      "DEV_Spk-000CDL:Cryo-PT-91_iDB" (EPICSToPLCLength:=15,
      EPICSToPLCDataBlockOffset:=572,
      PLCToEPICSLength:=25,
      PLCToEPICSDataBlockOffset:=1327);

        //********************************************
        // Device name: Spk-000CDL:Cryo-PT-92
        // Device type: ICS_PT_mbar
        //********************************************

      "DEV_Spk-000CDL:Cryo-PT-92_iDB" (EPICSToPLCLength:=15,
      EPICSToPLCDataBlockOffset:=587,
      PLCToEPICSLength:=25,
      PLCToEPICSDataBlockOffset:=1352);

        //********************************************
        // Device name: Spk-000CDL:Cryo-PT-93
        // Device type: ICS_PT_mbar
        //********************************************

      "DEV_Spk-000CDL:Cryo-PT-93_iDB" (EPICSToPLCLength:=15,
      EPICSToPLCDataBlockOffset:=602,
      PLCToEPICSLength:=25,
      PLCToEPICSDataBlockOffset:=1377);

        //********************************************
        // Device name: Spk-000CDL:Cryo-PT-94
        // Device type: ICS_PT_mbar
        //********************************************

      "DEV_Spk-000CDL:Cryo-PT-94_iDB" (EPICSToPLCLength:=15,
      EPICSToPLCDataBlockOffset:=617,
      PLCToEPICSLength:=25,
      PLCToEPICSDataBlockOffset:=1402);

        //********************************************
        // Device name: Spk-000CDL:Cryo-PT-95
        // Device type: ICS_PT_mbar
        //********************************************

      "DEV_Spk-000CDL:Cryo-PT-95_iDB" (EPICSToPLCLength:=15,
      EPICSToPLCDataBlockOffset:=632,
      PLCToEPICSLength:=25,
      PLCToEPICSDataBlockOffset:=1427);

        //********************************************
        // Device name: Spk-000CDL:Vac-VGC-071
        // Device type: ICS_PT_mbar
        //********************************************

      "DEV_Spk-000CDL:Vac-VGC-071_iDB" (EPICSToPLCLength:=15,
      EPICSToPLCDataBlockOffset:=647,
      PLCToEPICSLength:=25,
      PLCToEPICSDataBlockOffset:=1452);

        //********************************************
        // Device name: Spk-000CDL:Vac-VGP-070
        // Device type: ICS_PT_mbar
        //********************************************

      "DEV_Spk-000CDL:Vac-VGP-070_iDB" (EPICSToPLCLength:=15,
      EPICSToPLCDataBlockOffset:=662,
      PLCToEPICSLength:=25,
      PLCToEPICSDataBlockOffset:=1477);
END_FUNCTION
DATA_BLOCK "EPICS_DebuggerResult"
{ S7_Optimized_Access := 'TRUE' }
VERSION : 0.1
NON_RETAIN
   VAR
      EPICS_Debugger_UtilitiesCall : String;   // PLCFactory Utilities call status
      EPICS_Debugger_DeviceCalls : String;   // PLCFactory DeviceCalls status
      EPICS_Debugger_IOCHash : String;   // EPICS IOC Hash vs. PLCFactory Hash
      EPICS_Debugger_ModBusHeartBeat : String;   // EPICS IOC Modbus (IOC->PLC) communication status
      EPICS_Debugger_S7Connection : String;   // EPICS IOC S7 TCP (PLC->IOC) communication status
      EPICS_Debugger_EPICS_GeneralState : String;   // Main status of the EPICS IOC communication
      EPICS_S7Port : Int;   // Actual TCP port that has been opened by the PLC
      EPICS_ModbusPort : Int;   // Actual ModBusTCP port that has been opened by the PLC
      EPICS_PLC_EthernetInterface : UInt;   // The currently used HW Identifer of the Ethernet Port on the PLC dedicated to EPICS
      EPICS_PayloadSize_InBytes : UInt;   // The currently configured payload size in bytes
      EPICS_PLC_Hash : DInt;   // The PLC Hash
      EPICS_PLCFactory_Version : String;   // The PLCFactory version that was used to generate the PLC code
      EPICS_CommunicationOK : Bool;   // Overall EPICS communication is OK
   END_VAR

BEGIN

END_DATA_BLOCK
FUNCTION_BLOCK "EPICS_DebuggerFB"
{ S7_Optimized_Access := 'TRUE' }
VERSION : 0.1
   VAR
      CheckUtilitiesTON {OriginalPartName := 'IEC_TIMER'; LibVersion := '1.0'; ExternalAccessible := 'False'; ExternalVisible := 'False'; ExternalWritable := 'False'} : TON_TIME;
      UtilSquareErrorTON { ExternalAccessible := 'False'; ExternalVisible := 'False'; ExternalWritable := 'False'} : Bool;
      CheckUtilitiesTON2 {OriginalPartName := 'IEC_TIMER'; LibVersion := '1.0'; ExternalAccessible := 'False'; ExternalVisible := 'False'; ExternalWritable := 'False'} : TON_TIME;
      UtilSquareErrorTON2 { ExternalAccessible := 'False'; ExternalVisible := 'False'; ExternalWritable := 'False'} : Bool;
      ModBus_TON {OriginalPartName := 'IEC_TIMER'; LibVersion := '1.0'; ExternalAccessible := 'False'; ExternalVisible := 'False'; ExternalWritable := 'False'} : TON_TIME;
      ModBus_wordsave { ExternalAccessible := 'False'; ExternalVisible := 'False'; ExternalWritable := 'False'} : Word;
   END_VAR
   VAR DB_SPECIFIC
      Helper_String { ExternalAccessible := 'False'; ExternalVisible := 'False'; ExternalWritable := 'False'} : String;
      Helper_String_Array { ExternalAccessible := 'False'; ExternalVisible := 'False'; ExternalWritable := 'False'} AT Helper_String : Struct
         String_Maximal { ExternalAccessible := 'False'; ExternalVisible := 'False'; ExternalWritable := 'False'} : Byte;
         String_Actual { ExternalAccessible := 'False'; ExternalVisible := 'False'; ExternalWritable := 'False'} : Byte;
         StringValueArray { ExternalAccessible := 'False'; ExternalVisible := 'False'; ExternalWritable := 'False'} : Array[0..15] of Byte;
      END_STRUCT;
   END_VAR
   VAR
      S7ConnTON {OriginalPartName := 'IEC_TIMER'; LibVersion := '1.0'; ExternalAccessible := 'False'; ExternalVisible := 'False'; ExternalWritable := 'False'} : TON_TIME;
   END_VAR

   VAR_TEMP
      AllOK { ExternalAccessible := 'False'; ExternalVisible := 'False'; ExternalWritable := 'False'} : Bool;
      i : Int;
      ModBusOK : Bool;
      S7OK : Bool;
   END_VAR


BEGIN
	//Author: Miklos Boros (miklos.boros@esss.se), Copyrigth 2017-2020 by European Spallation Source, Lund
	//This block was generated by PLCFactory
	//Description: This FB checks the EPICS configuration and outputs the result into EPICS_DebuggerResult.

	//DO NOT Modify this block!!!

	//AllOK will be evaluated in this code and passed to the EPICS_CommunicationOK signal that can be used by the PLC logic
	#AllOK := TRUE;

	#CheckUtilitiesTON(IN:="Utilities".Square_100ms,
	                   PT:=T#200ms,
	                   Q=>#UtilSquareErrorTON);

	#CheckUtilitiesTON2(IN := NOT "Utilities".Square_100ms,
	                   PT := T#200ms,
	                   Q => #UtilSquareErrorTON2);


	#ModBus_TON(IN := #ModBus_wordsave = "EPICSToPLC"."Word"[2],
	            PT := T#5s);


     "EPICS_DebuggerResult".#EPICS_PayloadSize_InBytes := 3004;
     "EPICS_DebuggerResult".#EPICS_PLC_Hash := 457744924;
     "EPICS_DebuggerResult".#EPICS_PLCFactory_Version := 'fb3b582a9a66e37ff877560bc4f23ab7654f4230';

	IF ("Utilities".AlwaysOn = FALSE) THEN
	    "EPICS_DebuggerResult".#EPICS_Debugger_UtilitiesCall := 'ERROR: FunctionBlock: "_UilitiesFB" is called with a wrong InstanceDB. Call it with the existing iDB named: "Utilities" AND check if the System Memory bits and the System Clock byte is enabled!';
         #AllOK := FALSE;
	ELSE
	    IF (#UtilSquareErrorTON OR #UtilSquareErrorTON2) THEN
	        "EPICS_DebuggerResult".#EPICS_Debugger_UtilitiesCall := 'ERROR: FunctionBlock: "_UilitiesFB" is called with a wrong InstanceDB. Call it with the existing iDB named: "Utilities" AND check if the System Memory bits and the System Clock byte is enabled!';
             #AllOK := FALSE;
	    ELSE
	        "EPICS_DebuggerResult".#EPICS_Debugger_UtilitiesCall := 'OK: EPICS Utilities works as expected.';

	    END_IF;
	END_IF;

	IF ("Utilities".EPICS_Device_calls_precessed) THEN
	    "EPICS_DebuggerResult".#EPICS_Debugger_DeviceCalls := 'OK: "EPICS_device_calls" is called as expected.';
	ELSE
	    "EPICS_DebuggerResult".#EPICS_Debugger_DeviceCalls := 'ERROR: "EPICS_device_calls" is not called in OB1!';
         #AllOK := FALSE;
	END_IF;

	IF (("EPICSToPLC"."Word"[0] = "PLCToEPICS"."Word"[0]) AND ("EPICSToPLC"."Word"[1] = "PLCToEPICS"."Word"[1])) THEN
	    "EPICS_DebuggerResult".#EPICS_Debugger_IOCHash := 'OK: IOC and PLC hash are equal.';
	ELSE
	    "EPICS_DebuggerResult".#EPICS_Debugger_IOCHash := 'ERROR: IOC and PLC hash are NOT equal!';
         #AllOK := FALSE;
	END_IF;

	IF (#ModBus_TON.Q) THEN
	    "EPICS_DebuggerResult".#EPICS_Debugger_ModBusHeartBeat := 'ERROR: The IOC is not sending any HeartBeat via ModBus!';
         #AllOK := FALSE;
	    #ModBusOK := FALSE;
	ELSE
	    "EPICS_DebuggerResult".#EPICS_Debugger_ModBusHeartBeat := 'OK: ModBus HeartBeat is received as expected.';
	    #ModBusOK := TRUE;
	END_IF;

	#S7ConnTON(IN := NOT "_CommsPLC_EPICS_DB".SendDone, PT := T#3s);

	IF ("_CommsPLC_EPICS_DB".BytesToSend > 0) THEN

	    IF (#S7ConnTON.Q) THEN
	        "EPICS_DebuggerResult".EPICS_Debugger_S7Connection := 'ERROR: EPICS S7 connection can not send Status variables!';
	        #S7OK := FALSE;
             #AllOK := FALSE;
	    ELSE
	        "EPICS_DebuggerResult".EPICS_Debugger_S7Connection := 'OK: EPICS S7 works as expected.';
	        #S7OK := TRUE;

	    END_IF;
	ELSE
	    "EPICS_DebuggerResult".EPICS_Debugger_S7Connection := 'OK: EPICS S7 disabled, there is no Status variable to send.';
	    #S7OK := TRUE;
	END_IF;

	IF (#ModBusOK AND #S7OK) THEN
	    "EPICS_DebuggerResult".EPICS_Debugger_EPICS_GeneralState := 'OK. EPICS IOC communication is ONLINE.';
	END_IF;

	IF (#ModBusOK AND NOT #S7OK) THEN
	    "EPICS_DebuggerResult".EPICS_Debugger_EPICS_GeneralState := 'ERROR. ModBus seems to be working but S7 TCP is blocked. Try to check your PLC router IP.';
         #AllOK := FALSE;
	END_IF;

	IF (NOT #ModBusOK AND #S7OK) THEN
	    "EPICS_DebuggerResult".EPICS_Debugger_EPICS_GeneralState := 'ERROR. ModBus seems to be offline. Waiting for IOC to finish connecting to the PLC.';
         #AllOK := FALSE;
	END_IF;

	IF ( NOT #ModBusOK AND NOT #S7OK) THEN
	    "EPICS_DebuggerResult".EPICS_Debugger_EPICS_GeneralState := 'ERROR. Both ModBus and S7 TCP seems to be offline. Check if your IOC is running and if it is connected to the right PLC interface. Your HardwareID comes from CCDB!';
         #AllOK := FALSE;
	END_IF;

	"EPICS_DebuggerResult".EPICS_ModbusPort := "_CommsPLC_EPICS_DB".MBPort;
	"EPICS_DebuggerResult".EPICS_S7Port := "_CommsPLC_EPICS_DB".S7Port;
	"EPICS_DebuggerResult".EPICS_PLC_EthernetInterface :=  "_CommsPLC_EPICS_DB".InterfaceID;

	#ModBus_wordsave := "EPICSToPLC"."Word"[2];

	//Put the Overall result to the Globl DB
	"EPICS_DebuggerResult".EPICS_CommunicationOK := #AllOK;


END_FUNCTION_BLOCK
DATA_BLOCK "EPICS_DebuggerFB_iDB"
{ S7_Optimized_Access := 'TRUE' }
VERSION : 0.1
NON_RETAIN
"EPICS_DebuggerFB"

BEGIN

END_DATA_BLOCK
ORGANIZATION_BLOCK "EPICS_DebuggerOB"
TITLE = "Main Program Sweep (Cycle)"
{ S7_Optimized_Access := 'TRUE' }
VERSION : 0.1

BEGIN
	//Author: Miklos Boros (miklos.boros@esss.se), Copyrigth 2017-2020 by European Spallation Source, Lund
	//This block was generated by PLCFactory
	//Description: This OB is a cyclic OB called in every PLC cycle and EPICS_DebuggerFB checks the EPICS configuration.

	//DO NOT Modify this block!!!
	"EPICS_DebuggerFB_iDB"();


END_ORGANIZATION_BLOCK
TYPE "typeModul"
VERSION : 0.1
   STRUCT
      slotLaddr : HW_IO;   // Hardware ID of  module
      slotErrorState : Bool;   // error state of module
   END_STRUCT;

END_TYPE


TYPE "typeDevice"
VERSION : 0.1
   STRUCT
      laddr : HW_DEVICE;   // Logical address of a device or slave (system constant in HW configuration)
      "name" : String[50];   // Device name
      errorState : USInt;   // Status of the device 1=ok!, 2=faulty, 3=lost connection, 4=disabled, 12= was faulty, 13=was lost, 14=was disabled
      error : Bool;   // Signalizes an error in the device/slave
      nextDevice : Int;   // device number of next device
      actualConfiguredModules : Int;   // Actual number of configured modules in the device
      slot : Array[0..30] of "typeModul";   // slot informations
   END_STRUCT;

END_TYPE


TYPE "typeIoSystem"
VERSION : 0.1
   STRUCT
      ioSystemId : UInt;   // ID of  IO System
      ioSystemError : Bool;   // TRUE: if an error is occured in the assigned IO System
      firstDevice : Int := 0;   // device number (index) of first device in IO System
      lastDevice : Int := 0;   // device number (index) of last device IO System
      actualConfiguredDevices : Int := 0;   // Actual number of configured devices in the IO System
      device : Array[1..60] of "typeDevice";   // List of all devices in the IO System
   END_STRUCT;

END_TYPE

TYPE "typePlc"
VERSION : 0.1
   STRUCT
      actualConfiguredCentralModules : Int;   // Actual number of configured local modules
      errorState : Bool;   // Status of the device 1=ok!, 2=faulty, 3=lost connection, 4=disabled, 12= was faulty, 13=was lost, 14=was disabled
      slot : Array[1..30] of "typeModul";   // slot informations
   END_STRUCT;

END_TYPE



DATA_BLOCK "DiagnosticsData"
TITLE = Diagosis data DB
{ S7_Optimized_Access := 'TRUE' }
AUTHOR : SIEMENS
FAMILY : Diagnose
NAME : '10'
VERSION : 0.1
NON_RETAIN
//The global data block contains the data structure of the IO system, the control, the devices with the modules and an error buffer.
   VAR
      plc { ExternalAccessible := 'True'; ExternalVisible := 'False'; ExternalWritable := 'False'; } : "typePlc";   // diagnosis information PLC
      ioSystem { ExternalAccessible := 'True'; ExternalVisible := 'False'; ExternalWritable := 'False'; } : Array[1..5] of "typeIoSystem";   // diagnosis information IO systems
   END_VAR


BEGIN

END_DATA_BLOCK

FUNCTION_BLOCK "DiagStartupIoSystem"
{ S7_Optimized_Access := 'TRUE' }
VERSION : 0.1
   VAR_INPUT DB_SPECIFIC
      ioSystemHwId { ExternalAccessible := 'True'; ExternalVisible := 'False'; ExternalWritable := 'False'; } : HW_IOSYSTEM;   // This ID is representing the IO System (PN or DP), find the ID in the system constants
   END_VAR

   VAR_OUTPUT
      status { ExternalAccessible := 'True'; ExternalVisible := 'False'; ExternalWritable := 'False'; } : Int;   // The return value of system function, where the last error occured
      instructionError { ExternalAccessible := 'True'; ExternalVisible := 'False'; ExternalWritable := 'False'; } : Int;   // Indicates in which system function the error occured: 1= DeviceStates PN , 2=GetName PN, 3=ModuleStates PN,  4=DeviceStates DP, 5= GetName DP. 6= ModuleStates DP
      errorIndex { ExternalAccessible := 'True'; ExternalVisible := 'False'; ExternalWritable := 'False'; } : Int;   // The last index of the respective loop, if an error occures
   END_VAR

   VAR_IN_OUT
      ioSystem : "typeIoSystem";   // The diagnostics structure for one IO System
   END_VAR

   VAR
      statActualConfiguredDevices { ExternalAccessible := 'True'; ExternalVisible := 'False'; ExternalWritable := 'False'; } : Int := 0;   // Actual number of devices in the PN IO System
      statGeoAddr {OriginalPartName := 'GEOADDR'; LibVersion := '1.0'; ExternalAccessible := 'True'; ExternalVisible := 'False'; ExternalWritable := 'False';} : GEOADDR;   // Slot information
      statGeoLaddr { ExternalAccessible := 'False'; ExternalVisible := 'False'; ExternalWritable := 'False'; } : HW_ANY;   // GEO2LOG hardware identifier
      statConfiguredDevices { ExternalAccessible := 'True'; ExternalVisible := 'False'; ExternalWritable := 'False'; } : Array[0..1023] of Bool;   // Temporary storage of the return of "DeviceStates", to combine the states of the devices with numbers and names
      statExistingDevices { ExternalAccessible := 'True'; ExternalVisible := 'False'; ExternalWritable := 'False'; } : Array[0..1023] of Bool;   // Temporary storage of the return of "DeviceStates", to combine the states of the devices with numbers and names
      statFaultyDevices { ExternalAccessible := 'True'; ExternalVisible := 'False'; ExternalWritable := 'False'; } : Array[0..1023] of Bool;   // Temporary storage of the return of "DeviceStates", to combine the states of the divices with numbers and names
      statDisabledDevices { ExternalAccessible := 'True'; ExternalVisible := 'False'; ExternalWritable := 'False'; } : Array[0..1023] of Bool;   // Storage of the status of all devices in the PN IO System --> State: Disabled
      statProblemDevices { ExternalAccessible := 'True'; ExternalVisible := 'False'; ExternalWritable := 'False'; } : Array[0..1023] of Bool;   // Storage of the status of all devices in the PN IO System --> State: Problem
      statDeviceModuleStates { ExternalAccessible := 'True'; ExternalVisible := 'False'; ExternalWritable := 'False'; } : Array[0..127] of Bool;   // Storage of the status of all modules in the PN Devices --> State: Problem
      instGetNameDevices {OriginalPartName := 'FB_806_S71500'; LibVersion := '1.3'; ExternalAccessible := 'True'; ExternalVisible := 'False'; ExternalWritable := 'False';} : Get_Name;   // Instance of system function "GetName"
      statInitString { ExternalAccessible := 'True'; ExternalVisible := 'False'; ExternalWritable := 'False'; } : String;   // Used to initialize the temporary string to convert into STRING[50]
      statFirstDevice { ExternalAccessible := 'True'; ExternalVisible := 'False'; ExternalWritable := 'False'; } : UInt;   // Station number of the first device of the list
      statFirstDeviceFlag { ExternalAccessible := 'False'; ExternalVisible := 'False'; ExternalWritable := 'False'; } : Bool := TRUE;   // Help tag for the first device in the linked list
      statLastDevice { ExternalAccessible := 'True'; ExternalVisible := 'False'; ExternalWritable := 'False'; } : UInt;   // Station number of the last device of the list
      statLinkedListPointer { ExternalAccessible := 'True'; ExternalVisible := 'False'; ExternalWritable := 'False'; } : Int;   // The actual index pointer of the linked list (Actual pointer = Station number of the device)
      statFirstRun { ExternalAccessible := 'False'; ExternalVisible := 'False'; ExternalWritable := 'False'; } : Bool := TRUE;   // Signalizes the first run
      statResetStatesOld { ExternalAccessible := 'True'; ExternalVisible := 'False'; ExternalWritable := 'False'; } : Bool;   // Detect a rising edge at ResetStates
      statMaxDevices { ExternalAccessible := 'True'; ExternalVisible := 'False'; ExternalWritable := 'False'; } : Int;
   END_VAR

   VAR_TEMP
      tempIndex : Int;   // index configured devices
      tempSlotIndex : Int;   // Loop index
      tempModuleNum : Int;   // index module number
      tempRetValGeo : Int;   // GEO2LOG error information
      tempRetValDeviceStates : Int;   // DeviceStates error information
      tempRetValModuleStates : Int;   // Return value system function ModuleStates
      tempStringConvert : String;   // Store the device names temporary here, to convert them into STRING[50]
      tempLastDevice : UInt;   // Temporary storage of the actual index, if it is the last device --> store it in static
      tempIoSystemError : Bool;
   END_VAR

   VAR CONSTANT
      STATE_CONFIGURED : USInt := 1;   // Used for instruction DeviceStates, read out all configured devices
      STATE_FAULTY : USInt := 2;   // Used for instruction DeviceStates, read out all faulty devices
      STATE_DISABLED : USInt := 3;   // Used for instruction DeviceStates, read out all disabled devices
      STATE_EXIST : USInt := 4;   // Used for instruction DeviceStates, read out all devices not reachable
      STATE_PROBLEM : USInt := 5;   // Used for instruction DeviceStates, read out all devices with several problems
      DEVICE_SLAVE : USInt := 2;   // GEO2LOG structure: HW type = 2
      MODULE_OF_DEVICE : USInt := 4;   // GEO2LOG structure: HW type = 4
      IO_SYSTEM_AREA : USInt := 1;   // GEO2LOG structure: Area = 1
      DP_SYSTEM_AREA : USInt := 2;   // GEO2LOG structure: Area = 2
      ERR_DEV_STATE_DEVICES : USInt := 1;   // Identifies the instruction behind the error code of output "Status" --> DeviceStates PN (Configured, faulty, existing)
      ERR_GET_NAME_DEVICES : USInt := 2;   // Identifies the instruction behind the error code of output "Status" -->  GetName of devices PN
      ERR_MOD_STAT_DEVICES : USInt := 3;   // Identifies the instruction behind the error code of output "Status" --> ModuleStates PN
      ERR_DEV_STAT_PN : USInt := 1;   // Value for output instruction error, DeviceStates PN devices
      ERR_MOD_STAT_PN : USInt := 4;   // Value for output instruction error, ModuleStates PN devices
      MAX_SLAVES_DP : Int := 127;
      MAX_SLAVES_PN : Int := 127;
   END_VAR


BEGIN
	//=============================================================================
	//Author: SIEMENS, Owner: Miklos Boros
	//        email: borosmiklos@gmail.com; miklos.boros@esss.se
	//
	//Functionality: Determine hardware identifier and module states from
	//               PN or DP IO system
	//
	//
	//Please Note:
	//        This block is part of the generated ESS Standard Code
	//        DON'T CHANGE THIS BLOCK MANUALY. Any changes will be overwritten in the next code generation.
	//
	//
	//Change log table:
	//Version  Date         Expert in charge      Changes applied
	//01.00.00 29.08.2017   ESS/ICS               First released version for PLCFactory
	//02.00.00 09-04-2018   ESS/ICS               Major bug fix for PN/DP devices
	//=============================================================================


	// The startup will be executed only once --> initialize the first run
	// indicator.
	#statFirstDeviceFlag := TRUE;
	#statFirstRun := TRUE;
	#statActualConfiguredDevices := 0;
	#statFirstDevice := 1;
	#statLastDevice := 1;

	//=============================================================================
	// CONFIGURED DEVICES
	//=============================================================================
	// Find out how much devices are configured in the IO System --> PROFINET IO
	// This number is the maximum number of devices, which will be checked in the
	// following programm
	#tempRetValDeviceStates := DeviceStates(LADDR := #ioSystemHwId,
	                                        MODE := #STATE_CONFIGURED,
	                                        STATE := #statConfiguredDevices);

	// Check if the block call was successful
	IF (#tempRetValDeviceStates <> 0)
	THEN
	    // Error handling
	    #status := #tempRetValDeviceStates;
	    #instructionError := #ERR_DEV_STATE_DEVICES;
	    // Call ok --> store the actual number of configured devices
	ELSE
	    ;
	END_IF;

	//=============================================================================
	// EXISTING DEVICES
	//=============================================================================
	#tempRetValDeviceStates := DeviceStates(LADDR := #ioSystemHwId,
	                                        MODE := #STATE_EXIST,
	                                        STATE := #statExistingDevices);

	// Check if the block call was successful
	IF (#tempRetValDeviceStates <> 0)
	THEN
	    // Error handling
	    #status := #tempRetValDeviceStates;
	    #instructionError := #ERR_DEV_STATE_DEVICES;
	    // Call ok --> store the actual number of configured devices
	ELSE
	    ;
	END_IF;

	//=============================================================================
	// FAULTY DEVICES
	//=============================================================================
	#tempRetValDeviceStates := DeviceStates(LADDR := #ioSystemHwId,
	                                        MODE := #STATE_FAULTY,
	                                        STATE := #statFaultyDevices);

	// Check if the block call was successful
	IF (#tempRetValDeviceStates <> 0)
	THEN
	    // Error handling
	    #status := #tempRetValDeviceStates;
	    #instructionError := #ERR_DEV_STATE_DEVICES;
	    // Call ok --> store the actual number of configured devices
	ELSE
	    ;
	END_IF;

	// Find out the number of the assigned IO system, to define if it is
	// a PN or DP Network
	#tempRetValGeo := LOG2GEO(LADDR := #ioSystemHwId,
	                          GEOADDR := #statGeoAddr);

	// set IO system ID
	#ioSystem.ioSystemId := #statGeoAddr.IOSYSTEM;

	// Inilize the structure for system function GEO2LOG
	#statGeoAddr.HWTYPE := #DEVICE_SLAVE;   // Hardware type 2: IO device
	// Predefine the type OF IO system. Either Profinet IO or Profibus DP
	IF ((#statGeoAddr.IOSYSTEM >= 100)
	    AND (#statGeoAddr.IOSYSTEM <= 115))
	THEN
	    #statGeoAddr.AREA := #IO_SYSTEM_AREA;   // Area ID 1: PROFINET IO
	    #statMaxDevices := #MAX_SLAVES_PN;
	ELSIF ((#statGeoAddr.IOSYSTEM >= 1)
	    AND (#statGeoAddr.IOSYSTEM <= 32))
	THEN
	    #statGeoAddr.AREA := #DP_SYSTEM_AREA;   // Area ID 1: Profibus DP
	    #statMaxDevices := #MAX_SLAVES_DP;
	ELSE
	    ;
	END_IF;

	// Go trough all devices and get the status of the configured
	FOR #tempIndex := 1 TO #statMaxDevices DO
	    // The devices are configured --> Read out the logical address and the
	    // device name
	    IF (#statConfiguredDevices[#tempIndex] = TRUE)
	    THEN
	        // Increment the actual configured devices, store the state and
	        // HW_ID as an numerical value (UINT)
	        #statActualConfiguredDevices := #statActualConfiguredDevices + 1;

	        // Store the first configured device for the linked list
	        IF (#statFirstDeviceFlag = TRUE)
	        THEN
	            #statFirstDevice := INT_TO_UINT(#tempIndex);
	            #ioSystem.firstDevice := UINT_TO_INT(#statFirstDevice);
	            #statFirstDeviceFlag := FALSE;
	            #tempLastDevice := INT_TO_UINT(#tempIndex);
	            // It is not the first bit --> Store the actual index as "next device"
	            // in the further one!
	        ELSE
	            #ioSystem.device[#tempLastDevice].nextDevice := #tempIndex;
	            #tempLastDevice := INT_TO_UINT(#tempIndex);
	        END_IF;
	        // Store the index of the last device for the exit condition of the
	        // followiing instructions
	        #statLastDevice := #tempLastDevice;
	        #ioSystem.lastDevice := UINT_TO_INT(#statLastDevice);

	        // Station number
	        #statGeoAddr.STATION := INT_TO_UINT(#tempIndex);
	        // read LADDR from devices
	        #tempRetValGeo := GEO2LOG(GEOADDR := #statGeoAddr,
	                                  LADDR => #statGeoLaddr);
	        // Everything is ok!
	        IF (#tempRetValGeo = 0)
	        THEN
	            // store LADDR from devices in diagnostic data block
	            #ioSystem.device[#tempIndex].laddr := #statGeoLaddr;

	            // Store the device name, if the device is existing
	            // Get name is an acyclic instruction. In the startup OB, the
	            // instruction has to be repeated until it is done or error
	            REPEAT
	                // Get device name of each decive in PN System
	                #instGetNameDevices(LADDR := #ioSystemHwId,
	                                    STATION_NR := #statGeoAddr.STATION,
	                                    DATA := #tempStringConvert);

	            UNTIL (#instGetNameDevices.DONE = TRUE)
	                OR (#instGetNameDevices.ERROR = TRUE)
	            END_REPEAT;

	            IF (#instGetNameDevices.ERROR = TRUE)
	            THEN
	                // Error handling
	                #status := WORD_TO_INT(#instGetNameDevices.STATUS);
	                #instructionError := #ERR_GET_NAME_DEVICES;
	                #errorIndex := #tempIndex;

	                // Everything is ok --> Convert the String[254] into String[50]
	            ELSIF (#instGetNameDevices.DONE = TRUE)
	            THEN
	                // Cut all characters more than 50 to reduce the string length
	                #ioSystem.device[#tempIndex].name := DELETE(IN := #tempStringConvert,
	                                                            L := 204,
	                                                            P := 50);

	                // Initialize the temporary string before next loop
	                #tempStringConvert := #statInitString;
	            ELSE
	                ;
	            END_IF;
	        ELSE
	            // If the return value ist not = 0 --> the device/system/module is
	            // not configured --> No error handling
	            // set LADDR from devices to 0 in diagnostic data block
	            #ioSystem.device[#tempIndex].laddr := 0;
	            #ioSystem.device[#tempIndex].name := '';
	        END_IF;

	        // Check if the configured devices are faulty or lost once through
	        // the startup!
	        IF (#statExistingDevices[#tempIndex] = TRUE)
	        THEN
	            IF (#statFaultyDevices[#tempIndex] = TRUE)
	            THEN

	                #ioSystem.device[#tempIndex].errorState := 2;
	                #ioSystem.device[#tempIndex].error := TRUE;

	                // The device is not faulty and does exist --> set state ok!
	            ELSE
	                #ioSystem.device[#tempIndex].errorState := 1;
	                #ioSystem.device[#tempIndex].error := FALSE;
	            END_IF;
	            // The connection to the device is lost at the moment
	        ELSE
	            #ioSystem.device[#tempIndex].errorState := 3;
	            #ioSystem.device[#tempIndex].error := TRUE;
	        END_IF;
	        // No device is configured
	    ELSE
	        ;
	    END_IF;

	END_FOR;
	// Store the actual configured devices in the diagnostics structure
	#ioSystem.actualConfiguredDevices := #statActualConfiguredDevices;

	// Mark parameter "Next Device" of the last device in the list
	// --> "Next Device" = negative --> Last device in the list
	#ioSystem.device[#statLastDevice].nextDevice := -1;

	// Go through the devices until the last device is reached
	// If there are gaps between the device-list, jump over and have a look on
	// the "NextDevice" parameter
	REPEAT
	    IF (#statFirstRun = TRUE)
	    THEN
	        // The index of the linked list is representing the station number.
	        #statGeoAddr.STATION := #statFirstDevice;
	        // Initialize the pointer for the first run
	        #statLinkedListPointer := UINT_TO_INT(#statFirstDevice);
	        // Reset the flag, which signalizes the first run.
	        #statFirstRun := FALSE;
	    ELSE
	        // The index of the linked list is representing the station number.
	        #statGeoAddr.STATION := INT_TO_UINT(#statLinkedListPointer);
	    END_IF;

	    //=============================================================================
	    // Get the logical address of all modules and store the actual number of
	    // modules from each device
	    //=============================================================================

	    // Inilize the structure for system function GEO2LOG
	    #statGeoAddr.HWTYPE := #MODULE_OF_DEVICE;   // Hardware type 4: Module
	    FOR #tempModuleNum := 0 TO 30 DO
	        // Slot number
	        #statGeoAddr.SLOT := INT_TO_UINT(#tempModuleNum);
	        // read LADDR from modules
	        #tempRetValGeo := GEO2LOG(GEOADDR := #statGeoAddr,
	                                  LADDR => #statGeoLaddr);
	        // check Retval
	        IF (#tempRetValGeo = 0)
	        THEN
	            // store LADDR from modules in diagnostic data block
	            #ioSystem.device[#statLinkedListPointer].slot[#tempModuleNum].slotLaddr := #statGeoLaddr;
	            #ioSystem.device[#statLinkedListPointer].actualConfiguredModules := #ioSystem.device[#statLinkedListPointer].actualConfiguredModules + 1;
	        ELSE
	            // If the return value ist not = 0 --> the device/system/module is
	            // not configured --> No error handling
	            // set LADDR from modules to 0 in diagnostic data block
	            #ioSystem.device[#statLinkedListPointer].slot[#tempModuleNum].slotLaddr := 0;
	        END_IF;
	    END_FOR;

	    //=============================================================================
	    // Check modules of faulty Devices
	    //=============================================================================

	    // Check the state of the configured devices
	    IF (#ioSystem.device[#statLinkedListPointer].errorState = 2)
	    THEN
	        // The device is reachable, but faulty because of an error in a
	        // subordinated system --> check the modules
	        #tempRetValModuleStates := ModuleStates(LADDR := #ioSystem.device[#statLinkedListPointer].laddr,
	                                                MODE := #STATE_PROBLEM,
	                                                STATE := #statDeviceModuleStates);

	        IF (#tempRetValModuleStates <> 0)
	        THEN
	            // Error hanlding
	            #status := #tempRetValModuleStates;
	            #instructionError := #ERR_MOD_STAT_DEVICES;
	            #errorIndex := UINT_TO_INT(#statFirstDevice);
	        ELSE
	            // Store the state of the different module in the diag DB
	            FOR #tempSlotIndex := 0 TO #ioSystem.device[#statFirstDevice].actualConfiguredModules DO
	                IF (#statDeviceModuleStates[#tempSlotIndex + 1] = TRUE)
	                THEN
	                    #ioSystem.device[#statLinkedListPointer].slot[#tempSlotIndex].slotErrorState := TRUE;
	                ELSE
	                    #ioSystem.device[#statLinkedListPointer].slot[#tempSlotIndex].slotErrorState := FALSE;
	                END_IF;
	            END_FOR;
	        END_IF;
	    ELSIF (#ioSystem.device[#statLinkedListPointer].errorState = 3)
	    THEN

	        FOR #tempSlotIndex := 0 TO #ioSystem.device[#statLinkedListPointer].actualConfiguredModules DO
	            IF (#ioSystem.device[#statLinkedListPointer].slot[#tempSlotIndex].slotLaddr <> 0)
	            THEN
	                #ioSystem.device[#statLinkedListPointer].slot[#tempSlotIndex].slotErrorState := TRUE;
	            END_IF;
	        END_FOR;

	    ELSE
	        ; // no faulty device --> nothing to do!
	    END_IF;

	    // Initialize the pointer for the next run
	    #statLinkedListPointer := #ioSystem.device[#statLinkedListPointer].nextDevice;
	    // If the last device is reached, reset the bit for the first run
	    //#FirstRun := TRUE;
	    // Checking the modules is done, the last device is reached
	UNTIL (#statLinkedListPointer < 0)
	END_REPEAT;
	// Reset the condition for the first run.
	#statFirstRun := TRUE;


END_FUNCTION_BLOCK

DATA_BLOCK "DiagStartupIoSystem_iDB"
{ S7_Optimized_Access := 'TRUE' }
VERSION : 0.1
NON_RETAIN
"DiagStartupIoSystem"

BEGIN

END_DATA_BLOCK

FUNCTION_BLOCK "DiagStartupPlc"
{ S7_Optimized_Access := 'TRUE' }
VERSION : 0.1
   VAR_OUTPUT
      status { ExternalAccessible := 'True'; ExternalVisible := 'False'; ExternalWritable := 'False'; } : Int;   // The return value of system function, where the last error occured
      instructionError { ExternalAccessible := 'True'; ExternalVisible := 'False'; ExternalWritable := 'False'; } : Int;   // Indicates in which system function the error occured: 1= DeviceStates PN , 2=GetName PN, 3=ModuleStates PN,  4=DeviceStates DP, 5= GetName DP. 6= ModuleStates DP
   END_VAR

   VAR_IN_OUT
      plc { ExternalAccessible := 'True'; ExternalVisible := 'False'; ExternalWritable := 'False'; } : "typePlc";   // The diagnostics structure for one PLC
   END_VAR

   VAR
      statGeoAddr {OriginalPartName := 'GEOADDR'; LibVersion := '1.0'; ExternalAccessible := 'False'; ExternalVisible := 'False'; ExternalWritable := 'False';} : GEOADDR;   // Slot information
      statGeoLaddr { ExternalAccessible := 'False'; ExternalVisible := 'False'; ExternalWritable := 'False'; } : HW_ANY;   // GEO2LOG hardware identifier
      statActualCentralModules { ExternalAccessible := 'True'; ExternalVisible := 'False'; ExternalWritable := 'False'; } : USInt := 0;   // Actual number of modules in the central station (PLC)
      statPlcModuleStates { ExternalAccessible := 'True'; ExternalVisible := 'False'; ExternalWritable := 'False'; } : Array[0..127] of Bool;   // Storage of the status of all modules in the PLC central station --> State: Problem
   END_VAR

   VAR_TEMP
      tempModuleNum : Int;   // index module number
      tempRetValGeo : Int;   // GEO2LOG error information
      tempRetValModuleStates : Int;   // Return value system function ModuleStates
   END_VAR

   VAR CONSTANT
      MODULE_OF_PLC : USInt := 4;   // GEO2LOG structure: HW type = 4
      CPU : USInt := 0;   // GEO2LOG structure: Area = 0
      CENTRAL_SYSTEM : USInt := 0;   // GEO2LOG structure: IO System = 0
      CENTRAL_STATION : USInt;   // GEO2LOG structure: Station = 0
      HW_ID_PLC_MODULES : HW_DEVICE := 32;   // HW ID of the PLC, which is needed for getting the module states --> fix value
      STATE_PROBLEM : USInt := 5;   // Used for instruction DeviceStates, read out all devices with several problems
      ERR_MOD_STAT_CENTRAL : USInt := 3;   // Value for output instruction error, ModuleStates local modules
   END_VAR


BEGIN
	//=============================================================================
	//Author: SIEMENS, Owner: Miklos Boros
	//        email: borosmiklos@gmail.com; miklos.boros@esss.se
	//
	//Functionality: Determine hardware identifier and module states from local
	//               modules
	//
	//
	//Please Note:
	//        This block is part of the generated ESS Standard Code
	//        DON'T CHANGE THIS BLOCK MANUALY. Any changes will be overwritten in the next code generation.
	//
	//
	//Change log table:
	//Version  Date         Expert in charge      Changes applied
	//01.00.00 29.08.2017   ESS/ICS               First released version for PLCFactory
	//02.00.00 09-04-2018   ESS/ICS               Major bug fix for PN/DP devices
	//=============================================================================


	//=============================================================================
	// Determine hardware identifier from LOCAL MODULES
	//=============================================================================
	#statGeoAddr.HWTYPE := #MODULE_OF_PLC;      // Hardware type 4: module
	#statGeoAddr.AREA := #CPU;                  // Area ID 0: CPU
	#statGeoAddr.IOSYSTEM := #CENTRAL_SYSTEM;   // PROFINET IO system
	                                            // (0 = central unit in the rack)
	#statGeoAddr.STATION := #CENTRAL_STATION;   // Number of the rack
	                                            // if area identifier
	                                            //  AREA = 0 (central module).

	FOR #tempModuleNum := 1 TO 30 DO
	  // Slot number
	  #statGeoAddr.SLOT := INT_TO_UINT(#tempModuleNum);
	  // read LADDR from local modules
	  #tempRetValGeo := GEO2LOG(GEOADDR := #statGeoAddr,
	                            LADDR => #statGeoLaddr);
	  // check Retval
	  IF (#tempRetValGeo = 0)
	  THEN
	    // store LADDR from local modules in diagnostic data block
	    #plc.slot[#tempModuleNum].slotLaddr := #statGeoLaddr;
	    #statActualCentralModules := #statActualCentralModules + 1;
	  ELSE
	    // If the return value ist not = 0 --> the device/system/module is not
	    // configured --> No error handling
	    // set LADDR from local modules to 0 in diagnostic data block
	    #plc.slot[#tempModuleNum].slotLaddr := 0;
	  END_IF;
	  // Store the actual configured devices in the diagnostics DB
	  #plc.actualConfiguredCentralModules := #statActualCentralModules;
	END_FOR;


	//=============================================================================
	// Check module states from LOCAL MODULES
	//=============================================================================
	// Check if central module are available - at least one module is always
	// configured, the PLC itself
	IF (#plc.actualConfiguredCentralModules > 1)
	THEN
	  // Check the status of the local modules
	  #tempRetValModuleStates := ModuleStates(LADDR := #HW_ID_PLC_MODULES,
	                                          MODE := #STATE_PROBLEM,
	                                          STATE := #statPlcModuleStates);

	  // Check if the block call was successful
	  IF (#tempRetValModuleStates <> 0)
	  THEN
	    // Error handling
	    #status := #tempRetValModuleStates;
	    #instructionError := #ERR_MOD_STAT_CENTRAL;
	  ELSE
	    ; // Everything is ok!
	  END_IF;
	ELSE
	  ; // There are no central module configured
	END_IF;

	// The error LED of the PLC is flashing --> Set error state of the PLC
	#plc.errorState := TRUE;


	//=============================================================================
	// set module states from LOCAL MODULES
	//=============================================================================

	// If the first bit in the array is true, at least one module is faulty
	IF (#statPlcModuleStates[0] = TRUE)
	THEN
	  // Check which of the modules are faulty
	  // PLC modules array starts at index 2 for the first local module
	  FOR #tempModuleNum := 2 TO #plc.actualConfiguredCentralModules + 1 DO
	    IF (#statPlcModuleStates[#tempModuleNum] = TRUE)
	    THEN
	      #plc.slot[#tempModuleNum - 1].slotErrorState := TRUE;
	    ELSE
	      #plc.slot[#tempModuleNum - 1].slotErrorState := FALSE;
	    END_IF;
	  END_FOR;

	ELSE
	  // Everything is ok!
	  FOR #tempModuleNum := 1 TO #plc.actualConfiguredCentralModules DO
	    #plc.slot[#tempModuleNum].slotErrorState := FALSE;
	  END_FOR;

	END_IF;

END_FUNCTION_BLOCK


DATA_BLOCK "DiagStartupPlc_iDB"
{ S7_Optimized_Access := 'TRUE' }
VERSION : 0.1
NON_RETAIN
"DiagStartupPlc"

BEGIN

END_DATA_BLOCK

FUNCTION "DiagnosticError" : Void
{ S7_Optimized_Access := 'TRUE' }
VERSION : 0.1
   VAR_INPUT
      ioState : Word;   // IO state of the HW object
      laddr : HW_ANY;   // Hardware identifier
      channel : UInt;   // Channel number
      multiError : Bool;   // =true if more than one error is present
   END_VAR

   VAR_IN_OUT
      plc : "typePlc";   // The diagnostics structure for one PLC
      ioSystem : Array[1..5] of "typeIoSystem";   // The diagnostics structure for one IO System
   END_VAR

   VAR_TEMP
      tempGeoAddr {OriginalPartName := 'GEOADDR'; LibVersion := '1.0'} : GEOADDR;   // Geographical address of the disturbed Module / Device
      tempIoSystemIndex : Int;   // Index for IO System
      index : Int;   // index system
      tempRetVal : Int;   // Return value of LOG2GEO
   END_VAR

   VAR CONSTANT
      GOOD : Word := 16#0001;   // Status of the hardware object: Bit 0: Good
      AREA_CENTRAL : UInt := 0;   // Area ID for PLC
      AREA_PROFINET : UInt := 1;   // Area ID for PROFINET IO
      AREA_PROFIBUS : UInt := 2;   // Area ID for PROFIBUS DP
   END_VAR


BEGIN
	//=============================================================================
	//Author: SIEMENS, Owner: Miklos Boros
	//        email: borosmiklos@gmail.com; miklos.boros@esss.se
	//
	//Functionality: Evaluate Diagnostic interrupt OB information for PLC and
	//               devices
	//
	//
	//Please Note:
	//        This block is part of the generated ESS Standard Code
	//        DON'T CHANGE THIS BLOCK MANUALY. Any changes will be overwritten in the next code generation.
	//
	//
	//Change log table:
	//Version  Date         Expert in charge      Changes applied
	//01.00.00 29-08-2017   ESS/ICS               First released version for PLCFactory
	//02.00.00 09-04-2018   ESS/ICS               Major bug fix for PN/DP devices
	//=============================================================================


	//=============================================================================
	// determine geographic address of faulty device
	//=============================================================================
	#tempRetVal := LOG2GEO(LADDR := #laddr,
	                       GEOADDR := #tempGeoAddr);


	//=============================================================================
	// evaluate diagnosis information for devices in an IO system
	//=============================================================================
	IF (#tempGeoAddr.AREA = #AREA_PROFINET)
	    OR (#tempGeoAddr.AREA = #AREA_PROFIBUS)
	THEN

	    //=============================================================================
	    // determine index for IO system
	    //=============================================================================
	    FOR #index := 1 TO 5 DO
	        IF ("DiagnosticsData".ioSystem[#index].ioSystemId = #tempGeoAddr.IOSYSTEM)
	        THEN
	            #tempIoSystemIndex := #index;
	        END_IF;
	    END_FOR;

	    IF (#tempIoSystemIndex <= 5)
	        AND (#tempGeoAddr.STATION <= 30)
	        AND (#tempGeoAddr.SLOT <= 30)
	    THEN
	        // evaluate diagnosis information IO system
	        IF (#ioState = #GOOD)
	        THEN
	            #ioSystem[#tempIoSystemIndex].device[#tempGeoAddr.STATION].error := FALSE;
	            #ioSystem[#tempIoSystemIndex].device[#tempGeoAddr.STATION].slot[#tempGeoAddr.SLOT].slotErrorState := FALSE;

	            IF (#ioSystem[#tempIoSystemIndex].device[#tempGeoAddr.STATION].errorState = 2)
	            THEN
	                #ioSystem[#tempIoSystemIndex].device[#tempGeoAddr.STATION].errorState := 12;
	            ELSIF (#ioSystem[#tempIoSystemIndex].device[#tempGeoAddr.STATION].errorState = 3)
	            THEN
	                #ioSystem[#tempIoSystemIndex].device[#tempGeoAddr.STATION].errorState := 13;
	            ELSE
	                #ioSystem[#tempIoSystemIndex].device[#tempGeoAddr.STATION].errorState := 1;
	            END_IF;
	        ELSE
	            #ioSystem[#tempIoSystemIndex].device[#tempGeoAddr.STATION].error := TRUE;
	            #ioSystem[#tempIoSystemIndex].device[#tempGeoAddr.STATION].errorState := 2;

	            #ioSystem[#tempIoSystemIndex].device[#tempGeoAddr.STATION].slot[#tempGeoAddr.SLOT].slotErrorState := TRUE;
	        END_IF;


	    END_IF;

	    //=============================================================================
	    // evaluate diagnosis information for PLC
	    //=============================================================================
	ELSIF (#tempGeoAddr.AREA = #AREA_CENTRAL)
	THEN

	    IF (#tempGeoAddr.SLOT <= 30)
	    THEN
	        // evaluate diagnosis information PLC
	        IF (#ioState = #GOOD)
	        THEN
	            #plc.slot[#tempGeoAddr.SLOT].slotErrorState := FALSE;
	        ELSE
	            #plc.slot[#tempGeoAddr.SLOT].slotErrorState := TRUE;
	        END_IF;

	    END_IF;

	ELSE
	    ;
	END_IF;

END_FUNCTION

FUNCTION "PullOrPlugModules" : Void
{ S7_Optimized_Access := 'TRUE' }
VERSION : 0.1
   VAR_INPUT
      laddr : HW_IO;   // Hardware identifier
      eventClass : Byte;   // 16#38/39: module inserted, removed
      faultId : Byte;   // Fault identifier
   END_VAR

   VAR_IN_OUT
      plc : "typePlc";   // The diagnostics structure for one PLC
      ioSystem : Array[1..5] of "typeIoSystem";   // The diagnostics structure for one IO System
   END_VAR

   VAR_TEMP
      tempIoSystemIndex : Int;   // Index for IO System
      index : Int;   // index system
      tempGeoAddr {OriginalPartName := 'GEOADDR'; LibVersion := '1.0'} : GEOADDR;   // Geographical address of the disturbed Module / Device
      tempRetVal : Int;   // Return value of LOG2GEO
   END_VAR

   VAR CONSTANT
      AREA_CENTRAL : UInt := 0;   // Area ID for PLC
      AREA_PROFINET : UInt := 1;   // Area ID for PROFINET IO
      AREA_PROFIBUS : UInt := 2;   // Area ID for PROFIBUS DP
      MODULE_PLUGGED : Byte := 16#38;   // (Sub)module plugged
      MODULE_PULLED : Byte := 16#39;   // (Sub)module pulled or not responding
      MODULE_MATCHES : Byte := 16#54;   // IO submodule inserted and matches configured submodule
      MODULE_OK : Byte := 16#61;   // Module inserted, module type OK
   END_VAR


BEGIN
	//=============================================================================
	//Author: SIEMENS, Owner: Miklos Boros
	//        email: borosmiklos@gmail.com; miklos.boros@esss.se
	//
	//Functionality: Evaluate Pull/plug interrupt OB information for PLC and
	//               devices
	//
	//
	//Please Note:
	//        This block is part of the generated ESS Standard Code
	//        DON'T CHANGE THIS BLOCK MANUALY. Any changes will be overwritten in the next code generation.
	//
	//
	//Change log table:
	//Version  Date         Expert in charge      Changes applied
	//01.00.00 29.08.2017   ESS/ICS               First released version for PLCFactory
	//02.00.00 09-04-2018   ESS/ICS               Major bug fix for PN/DP devices
	//=============================================================================


	//=============================================================================
	// determine geographic address of faulty device
	//=============================================================================
	#tempRetVal := LOG2GEO(LADDR := #laddr,
	                       GEOADDR := #tempGeoAddr);

	//=============================================================================
	// evaluate diagnosis information for devices in an IO system
	//=============================================================================
	IF (#tempGeoAddr.AREA = #AREA_PROFINET)
	    OR (#tempGeoAddr.AREA = #AREA_PROFIBUS)
	THEN

	    //=============================================================================
	    // determine index for IO system
	    //=============================================================================
	    FOR #index := 1 TO 5 DO
	        IF (#ioSystem[#index].ioSystemId = #tempGeoAddr.IOSYSTEM)
	        THEN
	            #tempIoSystemIndex := #index;
	        END_IF;
	    END_FOR;

	    IF (#tempIoSystemIndex <= 5)
	        AND (#tempGeoAddr.STATION <= 30)
	        AND (#tempGeoAddr.SLOT <= 30)
	    THEN
	        // check modules plugged
	        IF (#eventClass = #MODULE_PLUGGED)
	        THEN
	            // reset error state only if the correct module is inserted
	            IF (#faultId = #MODULE_MATCHES)
	                OR (#faultId = #MODULE_OK)
	            THEN
	                #ioSystem[#tempIoSystemIndex].device[#tempGeoAddr.STATION].error := FALSE;
	                #ioSystem[#tempIoSystemIndex].device[#tempGeoAddr.STATION].slot[#tempGeoAddr.SLOT].slotErrorState := FALSE;

	                IF (#ioSystem[#tempIoSystemIndex].device[#tempGeoAddr.STATION].errorState = 2)
	                THEN
	                    #ioSystem[#tempIoSystemIndex].device[#tempGeoAddr.STATION].errorState := 12;
	                ELSIF (#ioSystem[#tempIoSystemIndex].device[#tempGeoAddr.STATION].errorState = 3)
	                THEN
	                    #ioSystem[#tempIoSystemIndex].device[#tempGeoAddr.STATION].errorState := 13;
	                ELSE
	                    #ioSystem[#tempIoSystemIndex].device[#tempGeoAddr.STATION].errorState := 1;
	                END_IF;
	            END_IF;

	            // check modules pulled
	        ELSIF (#eventClass = #MODULE_PULLED)
	        THEN
	            #ioSystem[#tempIoSystemIndex].device[#tempGeoAddr.STATION].error := TRUE;
	            #ioSystem[#tempIoSystemIndex].device[#tempGeoAddr.STATION].errorState := 2;

	            #ioSystem[#tempIoSystemIndex].device[#tempGeoAddr.STATION].slot[#tempGeoAddr.SLOT].slotErrorState := TRUE;

	        ELSE
	            ;
	        END_IF;


	    END_IF;

	    //=============================================================================
	    // evaluate diagnosis information for PLC
	    //=============================================================================
	ELSIF (#tempGeoAddr.AREA = #AREA_CENTRAL)
	THEN

	    IF (#tempGeoAddr.SLOT <= 30)
	    THEN
	        IF (#eventClass = #MODULE_PLUGGED)
	        THEN
	            IF (#faultId = #MODULE_MATCHES)
	                OR (#faultId = #MODULE_OK)
	            THEN
	                #plc.slot[#tempGeoAddr.SLOT].slotErrorState := FALSE;
	            END_IF;

	        ELSIF (#eventClass = #MODULE_PULLED)
	        THEN
	            #plc.slot[#tempGeoAddr.SLOT].slotErrorState := TRUE;
	        ELSE
	            ;
	        END_IF;


	    END_IF;

	ELSE
	    ;
	END_IF;

END_FUNCTION

FUNCTION "RackOrStationFaliure" : Void
{ S7_Optimized_Access := 'TRUE' }
VERSION : 0.1
   VAR_INPUT
      laddr : HW_DEVICE;   // Hardware identifier
      eventClass : Byte;   // Event class
      faultId : Byte;   // Fault identifier
   END_VAR

   VAR_IN_OUT
      plc : "typePlc";   // The diagnostics structure for one PLC
      ioSystem : Array[1..5] of "typeIoSystem";   // The diagnostics structure for one IO System
   END_VAR

   VAR_TEMP
      index : Int;   // index system
      tempSlotIndex : Int;   // Loop index
      tempIoSystemIndex : Int;   // Index for IO System
      tempGeoAddr {OriginalPartName := 'GEOADDR'; LibVersion := '1.0'} : GEOADDR;   // Geographical address of the disturbed Module / Device
      tempRetVal : Int;   // Return value of LOG2GEO
      tempRetValModuleStates : Int;   // Return value system function ModuleStates
      tempDeviceModuleStates : Array[0..127] of Bool;   // Storage of the status of all modules in the PN Devices --> State: Problem
      tempLaddr : HW_DEVICE;   // logical address of the disturbed Module / Device
   END_VAR

   VAR CONSTANT
      AREA_CENTRAL : UInt := 0;   // Area ID for PLC
      AREA_PROFINET : UInt := 1;   // Area ID for PROFINET IO
      AREA_PROFIBUS : UInt := 2;   // Area ID for PROFIBUS DP
      SLAVE_DEVICE_RET : Byte := 16#38;   // return of a DP slave / IO device
      SLAVE_DEVICE_FAIL : Byte := 16#39;   // Failure of a DP slave / IO device
      DP_SLAVE_FAIL_RET : Byte := 16#C4;   // Failure/return of a DP slave
      IO_DEVICE_FAIL_RET : Byte := 16#CB;   // Failure/return of a PROFINET IO device
      STATE_PROBLEM : USInt := 5;   // Used for instruction DeviceStates, read out all devices with several problems
   END_VAR


BEGIN
	//=============================================================================
	//Author: SIEMENS, Owner: Miklos Boros
	//        email: borosmiklos@gmail.com; miklos.boros@esss.se
	//
	//Functionality: Evaluate Rack/Station interrupt OB information for PLC and
	//               devices
	//
	//
	//Please Note:
	//        This block is part of the generated ESS Standard Code
	//        DON'T CHANGE THIS BLOCK MANUALY. Any changes will be overwritten in the next code generation.
	//
	//
	//Change log table:
	//Version  Date         Expert in charge      Changes applied
	//01.00.00 29.08.2017   ESS/ICS               First released version for PLCFactory
	//02.00.00 09-04-2018   ESS/ICS               Major bug fix for PN/DP devices
	//=============================================================================


	//=============================================================================
	// determine geographic address of faulty device
	//=============================================================================
	#tempRetVal := LOG2GEO(LADDR := #laddr,
	                       GEOADDR := #tempGeoAddr);

	//=============================================================================
	// evaluate diagnosis information for devices in an IO system
	//=============================================================================
	IF (#tempGeoAddr.AREA = #AREA_PROFINET)
	  OR (#tempGeoAddr.AREA = #AREA_PROFIBUS)
	THEN

	  //===========================================================================
	  // determine index for IO system
	  //===========================================================================
	  FOR #index := 1 TO 5 DO
	    IF (#ioSystem[#index].ioSystemId = #tempGeoAddr.IOSYSTEM)
	    THEN
	      #tempIoSystemIndex := #index;
	    END_IF;
	  END_FOR;

	  IF (#tempIoSystemIndex <= 5)
	    AND (#tempGeoAddr.STATION <= 30)
	    AND (#tempGeoAddr.SLOT <= 30)
	  THEN
	    // check DP slave or IO device return
	    IF (#eventClass = #SLAVE_DEVICE_RET)
	    THEN
	      // reset error state only if the slave or device state is OK
	      IF (#faultId = #DP_SLAVE_FAIL_RET)
	        OR (#faultId = #IO_DEVICE_FAIL_RET)
	      THEN
	        #ioSystem[#tempIoSystemIndex].device[#tempGeoAddr.STATION].error := FALSE;

	        FOR #tempSlotIndex := 0 TO #ioSystem[#tempIoSystemIndex].device[#tempGeoAddr.STATION].actualConfiguredModules DO
	          #ioSystem[#tempIoSystemIndex].device[#tempGeoAddr.STATION].slot[#tempSlotIndex].slotErrorState := FALSE;
	        END_FOR;

	        IF (#ioSystem[#tempIoSystemIndex].device[#tempGeoAddr.STATION].errorState = 2)
	        THEN
	          #ioSystem[#tempIoSystemIndex].device[#tempGeoAddr.STATION].errorState := 12;
	        ELSIF (#ioSystem[#tempIoSystemIndex].device[#tempGeoAddr.STATION].errorState = 3)
	        THEN
	          #ioSystem[#tempIoSystemIndex].device[#tempGeoAddr.STATION].errorState := 13;
	        ELSE
	          #ioSystem[#tempIoSystemIndex].device[#tempGeoAddr.STATION].errorState := 1;
	        END_IF;

	      ELSE

	        // The device is reachable, but faulty because of an error in a
	        // subordinated system --> check the modules
	        #tempRetVal := GEO2LOG(LADDR => #tempLaddr,
	                               GEOADDR := #tempGeoAddr);

	        #tempRetValModuleStates := ModuleStates(LADDR := #tempLaddr,
	                                                MODE := #STATE_PROBLEM,
	                                                STATE := #tempDeviceModuleStates);

	        IF (#tempRetValModuleStates = 0)
	        THEN
	          // Store the state of the different module in the diag DB
	          FOR #tempSlotIndex := 0 TO #ioSystem[#tempIoSystemIndex].device[#tempGeoAddr.STATION].actualConfiguredModules DO
	            IF (#tempDeviceModuleStates[#tempSlotIndex + 1] = TRUE)
	            THEN
	              #ioSystem[#tempIoSystemIndex].device[#tempGeoAddr.STATION].slot[#tempSlotIndex].slotErrorState := TRUE;
	            ELSE
	              #ioSystem[#tempIoSystemIndex].device[#tempGeoAddr.STATION].slot[#tempSlotIndex].slotErrorState := FALSE;
	            END_IF;
	          END_FOR;
	        END_IF;

	        #ioSystem[#tempIoSystemIndex].device[#tempGeoAddr.STATION].errorState := 2;

	      END_IF;

	      // check DP slave or IO device failure
	    ELSIF (#eventClass = #SLAVE_DEVICE_FAIL)
	    THEN
	      #ioSystem[#tempIoSystemIndex].device[#tempGeoAddr.STATION].error := TRUE;
	      #ioSystem[#tempIoSystemIndex].device[#tempGeoAddr.STATION].errorState := 3;

	      FOR #tempSlotIndex := 0 TO #ioSystem[#tempIoSystemIndex].device[#tempGeoAddr.STATION].actualConfiguredModules DO
	        IF #ioSystem[#tempIoSystemIndex].device[#tempGeoAddr.STATION].slot[#tempSlotIndex].slotLaddr <> 0
	        THEN
	          #ioSystem[#tempIoSystemIndex].device[#tempGeoAddr.STATION].slot[#tempSlotIndex].slotErrorState := TRUE;
	        END_IF;
	      END_FOR;

	    ELSE
	      ;
	    END_IF;


	  END_IF;

	//=============================================================================
	//evaluate diagnosis information for PLC
	//=============================================================================
	ELSIF (#tempGeoAddr.AREA = #AREA_CENTRAL)
	THEN

	  IF (#tempGeoAddr.SLOT <= 30)
	  THEN
	    // check DP slave or IO device return
	    IF (#eventClass = #SLAVE_DEVICE_RET)
	    THEN
	      IF (#faultId = #DP_SLAVE_FAIL_RET)
	        OR (#faultId = #IO_DEVICE_FAIL_RET)
	      THEN
	        #plc.slot[#tempGeoAddr.SLOT].slotErrorState := FALSE;
	      END_IF;

	      // check DP slave or IO device failure
	    ELSIF (#eventClass = #SLAVE_DEVICE_FAIL)
	    THEN
	      #plc.slot[#tempGeoAddr.SLOT].slotErrorState := TRUE;
	    ELSE
	      ;
	    END_IF;


	  END_IF;

	ELSE
	  ;
	END_IF;

END_FUNCTION

FUNCTION_BLOCK "Diagnostics"
{ S7_Optimized_Access := 'TRUE' }
VERSION : 0.1
   VAR_IN_OUT
      plc { ExternalAccessible := 'True'; ExternalVisible := 'False'; ExternalWritable := 'False'; } : "typePlc";   // The diagnostics structure for one PLC
      ioSystem { ExternalAccessible := 'True'; ExternalVisible := 'False'; ExternalWritable := 'False'; } : Array[1..5] of "typeIoSystem";   // The diagnostics structure for one IO System
   END_VAR

   VAR
      statIoSystemIndex { ExternalAccessible := 'True'; ExternalVisible := 'False'; ExternalWritable := 'False'; } : Int;   // Index for IO System
      statSlotIndex { ExternalAccessible := 'True'; ExternalVisible := 'False'; ExternalWritable := 'False'; } : Int;   // Index for Slot
      statDeviceIndex { ExternalAccessible := 'True'; ExternalVisible := 'False'; ExternalWritable := 'False'; } : Int;   // Index for Device
   END_VAR

   VAR_TEMP
      retValLed : Int;
   END_VAR

   VAR CONSTANT
      ERROR_LED : UInt := 2;   // Identification number of the ERROR LED
      ERROR_LED_ON : UInt := 4;   // LED status Color 1 flashing
   END_VAR


BEGIN
	//=============================================================================
	//Author: SIEMENS, Owner: Miklos Boros
	//        email: borosmiklos@gmail.com; miklos.boros@esss.se
	//
	//Functionality: Basic diagnostic function that has to be called in every cycle
	//
	//
	//Please Note:
	//        This block is part of the generated ESS Standard Code
	//        DON'T CHANGE THIS BLOCK MANUALY. Any changes will be overwritten in the next code generation.
	//
	//
	//Change log table:
	//Version  Date         Expert in charge      Changes applied
	//01.00.00 29.08.2017   ESS/ICS               First released version for PLCFactory
	//02.00.00 09-04-2018   ESS/ICS               Major bug fix for PN/DP devices
	//=============================================================================


	//=============================================================================
	// check error active
	//=============================================================================
	#retValLed := LED(LADDR := "Local~Common", LED := #ERROR_LED);
	IF #retValLed = #ERROR_LED_ON
	THEN
	    #plc.errorState := TRUE;
	ELSE
	    #plc.errorState := FALSE;
	END_IF;

	//=============================================================================
	// check error in IO systems active
	//=============================================================================
	FOR #statIoSystemIndex := 1 TO 5 DO
	    #ioSystem[#statIoSystemIndex].ioSystemError := FALSE;

	    FOR #statDeviceIndex := 1 TO 60 DO
	        IF (#ioSystem[#statIoSystemIndex].device[#statDeviceIndex].error = TRUE)
	        THEN
	            #ioSystem[#statIoSystemIndex].ioSystemError := TRUE;
	        END_IF;
	    END_FOR;
	END_FOR;



END_FUNCTION_BLOCK

DATA_BLOCK "Diagnostics_iDB"
{ S7_Optimized_Access := 'TRUE' }
VERSION : 0.1
NON_RETAIN
"Diagnostics"

BEGIN

END_DATA_BLOCK

ORGANIZATION_BLOCK "CyclicDiagnostics"
TITLE = "Main Program Sweep (Cycle)"
{ S7_Optimized_Access := 'TRUE' }
VERSION : 0.1

BEGIN
	//=============================================================================
	//Author: SIEMENS, Owner: Miklos Boros
	//        email: borosmiklos@gmail.com; miklos.boros@esss.se
	//
	//Functionality: Main Cycle OB for diagnostics
	//               OB type: Program cycle
	//
	//
	//Please Note:
	//        This block is part of the generated ESS Standard Code
	//        DON'T CHANGE THIS BLOCK MANUALY. Any changes will be overwritten in the next code generation.
	//
	//
	//Change log table:
	//Version  Date         Expert in charge      Changes applied
	//01.00.00 29-08-2017   ESS/ICS               First released version for PLCFactory
	//02.00.00 09-04-2018   ESS/ICS               Major bug fix for PN/DP devices
	//=============================================================================



	"Diagnostics_iDB"(plc:="DiagnosticsData".plc,
	                  ioSystem:="DiagnosticsData".ioSystem);

END_ORGANIZATION_BLOCK


ORGANIZATION_BLOCK "Diagnostic error interrupt"
{ S7_Optimized_Access := 'TRUE' }
VERSION : 0.1

BEGIN
	//=============================================================================
	//Author: SIEMENS, Owner: Miklos Boros
	//        email: borosmiklos@gmail.com; miklos.boros@esss.se
	//
	//Functionality: Diagnostics Error Interrupt OB
	//               OB type: Diagnostic Interrupt
	//
	//
	//Please Note:
	//        This block is part of the generated ESS Standard Code
	//        DON'T CHANGE THIS BLOCK MANUALY. Any changes will be overwritten in the next code generation.
	//
	//
	//Change log table:
	//Version  Date         Expert in charge      Changes applied
	//01.00.00 29-08-2017   ESS/ICS               First released version for PLCFactory
	//02.00.00 09-04-2018   ESS/ICS               Major bug fix for PN/DP devices
	//=============================================================================

	//
	"DiagnosticError"(ioState:=#IO_State,
	                  laddr:=#LADDR,
	                  channel:=#Channel,
	                  multiError:=#MultiError,
	                  plc:="DiagnosticsData".plc,
	                  ioSystem:="DiagnosticsData".ioSystem);

END_ORGANIZATION_BLOCK

ORGANIZATION_BLOCK "Pull or plug of modules"
{ S7_Optimized_Access := 'TRUE' }
VERSION : 0.1

BEGIN
	//=============================================================================
	//Author: SIEMENS, Owner: Miklos Boros
	//        email: borosmiklos@gmail.com; miklos.boros@esss.se
	//
	//Functionality: Pull or Plug of mudules OB
	//               OB type: Pull or Plug of devices
	//
	//
	//Please Note:
	//        This block is part of the generated ESS Standard Code
	//        DON'T CHANGE THIS BLOCK MANUALY. Any changes will be overwritten in the next code generation.
	//
	//
	//Change log table:
	//Version  Date         Expert in charge      Changes applied
	//01.00.00 29-08-2017   ESS/ICS               First released version for PLCFactory
	//02.00.00 09-04-2018   ESS/ICS               Major bug fix for PN/DP devices
	//=============================================================================

	"PullOrPlugModules"(laddr:=#LADDR,
	                    eventClass:=#Event_Class,
	                    faultId:=#Fault_ID,
	                    plc:="DiagnosticsData".plc,
	                    ioSystem:="DiagnosticsData".ioSystem);

END_ORGANIZATION_BLOCK

ORGANIZATION_BLOCK "Rack or station failure"
{ S7_Optimized_Access := 'TRUE' }
VERSION : 0.1

BEGIN
	//=============================================================================
	//Author: SIEMENS, Owner: Miklos Boros
	//        email: borosmiklos@gmail.com; miklos.boros@esss.se
	//
	//Functionality: Rack or Station faliure OB
	//               OB type: Rack or station failure
	//
	//
	//Please Note:
	//        This block is part of the generated ESS Standard Code
	//        DON'T CHANGE THIS BLOCK MANUALY. Any changes will be overwritten in the next code generation.
	//
	//
	//Change log table:
	//Version  Date         Expert in charge      Changes applied
	//01.00.00 29-08-2017   ESS/ICS               First released version for PLCFactory
	//02.00.00 09-04-2018   ESS/ICS               Major bug fix for PN/DP devices
	//=============================================================================

	"RackOrStationFaliure"(laddr:=#LADDR,
	                       eventClass:=#Event_Class,
	                       faultId:=#Fault_ID,
	                       plc:="DiagnosticsData".plc,
	                       ioSystem:="DiagnosticsData".ioSystem);

END_ORGANIZATION_BLOCK

ORGANIZATION_BLOCK "Startup"
TITLE = "Complete Restart"
{ S7_Optimized_Access := 'TRUE' }
VERSION : 0.1

BEGIN
	//=============================================================================
	//Author: SIEMENS, Owner: Miklos Boros
	//        email: borosmiklos@gmail.com; miklos.boros@esss.se
	//
	//Functionality:
	//        This OB is a Startup OB, it will be called after OB100 and before the main cycle.
	//
	//
	//Please Note:
	//        This block is part of the generated ESS Standard Code however you should use
	//        the proper ioSystem ID from the
	//
	//Change log table:
	//Version  Date         Expert in charge      Changes applied
	//01.00.00 29.08.2017   ESS/ICS               First released version for PLCFactory
	//02.00.00 09-04-2018   ESS/ICS               Major bug fix for PN/DP devices
	//=============================================================================

	//Initialize the Main PLC Diagnostic
	"DiagStartupPlc_iDB"(plc:="DiagnosticsData".plc);


	//Put your current IO device configuration here. HW identifiers are in the PLC Tags/System constants!
	//Initialize IOSystem1
	//"DiagStartupIoSystem_iDB"(ioSystemHwId:=268,
	//                          ioSystem:="DiagnosticsData".ioSystem[1]);




END_ORGANIZATION_BLOCK

DATA_BLOCK "EPICSToPLC"
{ S7_Optimized_Access := 'FALSE' }
VERSION : 0.1
//########## EPICS->PLC datablock ##########
   STRUCT
      "Word" { ExternalAccessible := 'False'; ExternalVisible := 'False'; ExternalWritable := 'False'; } : Array[0..676] of Word;
   END_STRUCT;

BEGIN

END_DATA_BLOCK

DATA_BLOCK "PLCToEPICS"
{ S7_Optimized_Access := 'FALSE' }
VERSION : 0.1
NON_RETAIN
//########## PLC->EPICS datablock ##########
   STRUCT
      "Word" { ExternalAccessible := 'False'; ExternalVisible := 'False'; ExternalWritable := 'False'; } : Array[0..1501] of Word;
   END_STRUCT;

BEGIN

END_DATA_BLOCK

FUNCTION "_CommsEPICS" : Void
{ S7_Optimized_Access := 'TRUE' }
VERSION : 0.1
   VAR_TEMP
      PLC_Hash : DInt;
   END_VAR

BEGIN
	//Heartbeat PLC->EPICS
	IF "Utilities".Pulse_1s THEN
	    "PLCToEPICS"."Word"[2] := "PLCToEPICS"."Word"[2] + 1;
	    IF "PLCToEPICS"."Word"[2] >= 32000 THEN
	        "PLCToEPICS"."Word"[2] := 0;
	    END_IF;
	END_IF;

	// PLC Factory commit ID: fb3b582a9a66e37ff877560bc4f23ab7654f4230
	// PLC Hash (Generated by PLC Factory)
	#PLC_Hash := DINT#457744924;

	// Send the PLC Hash to the EPICS IOC
	"PLCToEPICS"."Word"[1] := DINT_TO_WORD(#PLC_Hash);
	"PLCToEPICS"."Word"[0] := DINT_TO_WORD(SHR(IN := #PLC_Hash, N := 16));

	// Send the PLC parameter upload status to the EPICS IOC
	"PLCToEPICS"."Word"[3] := "EPICSToPLC"."Word"[5];
     "Utilities".EPICSParametersStatus := "EPICSToPLC"."Word"[5];

	// Put the PLC Hash into the Modbus map
	"EPICSToPLC"."Word"[4] := DINT_TO_WORD(#PLC_Hash);
	"EPICSToPLC"."Word"[3] := DINT_TO_WORD(SHR(IN := #PLC_Hash, N := 16));


	// Put the payload size (in bytes) into the Modbus map
	"EPICSToPLC"."Word"[6] := 3004;

	// Call the comms block to provide PLC<->EPICS comms
	"_CommsPLC_EPICS_DB"(Enable         := "Utilities".AlwaysOn,
	                     SendTrigger    := "Utilities".Pulse_200ms,
	                     BytesToSend    := 3004,
	                     InterfaceID    := 72,
	                     S7ConnectionID := 256,
	                     MBConnectionID := 255,
	                     S7Port         := 2000,
	                     MBPort         := 502,
	                     PLCToEPICSData := "PLCToEPICS"."Word",
	                     EPICSToPLCData := "EPICSToPLC"."Word");

END_FUNCTION
